(* Logix 5000 project; controller DispersionPlc vendor 1 type 14 code 108 rev 34.11; software revision 34.01; part 13 of 22 *)
(* tags used below, declared in another part *)
   Estop_Disp : ALIAS FOR Local:3:I.Data.1;
   Estop_Inx : ALIAS FOR Local:3:I.Data.3;
   FC_4305_xx : AStd_PIDInterface;
   FCV_4305 : ALIAS FOR Local:13:O.Ch0Data;
   FIT_4305_xx : AStd_AnalogInput;
   FIT_4305_xx_AOI : AStd_AI_AOI;
   FIT_4305_xx_Holding : DINT;
   FIT_4305_xx_Samples : DINT;
   FV_4305_xx : AStd_VlvModulating;
   FV_4305_xx_AOI : AStd_VlVModulating_AOI;
   K400_PhaseTransfer : AStd_PLI;
   K400_PhaseTransfer_AOI : AStd_PLI_AOI;
   K400_PhaseTransfer_StepComplete : BOOL[32];
   LS_28_H : TIMER;
   LS_28_H_Alarm : BOOL;
   LS_4302_High : BOOL;
   P_4305 : AStd_FVNR;
   P_4305_AOI : AStd_FVNR_AOI;
   PUMP_P_4305_AUX : ALIAS FOR Local:1:I.Data[1].7;
   PUMP_P_4305_RUN : ALIAS FOR Local:1:O.Data[0].7;
   RO_HE4305_PhaseROHotWaterDrop : AStd_PLI;
   RO_HE4305_PhaseROHotWaterDrop_AOI : AStd_PLI_AOI;
   RO_HE4305_PhaseROWaterAddition : AStd_PLI;
   RO_Preheat_Temp : DINT;
   T4301_T4302_Xfer_In_Enable_Ctrl : BOOL;
   TC_4305_1 : AStd_PIDInterface;
   TC_4305_1_AOI : AStd_PIDInterface_AOI;
   TC_4305_1_PID : PID_ENHANCED;
   TCV_4305_1 : AStd_VlvModulating;
   TCV_4305_1_AOI : AStd_VlVModulating_AOI;
   TIT_4305_1 : AStd_AnalogInput;
   TIT_4305_1_AOI : AStd_AI_AOI;
   TIT_K400_1 : AStd_AnalogInput;
   TIT_K400_3 : AStd_AnalogInput;
   WIT_4302_1 : AStd_AnalogInput;
   XV_4301_8 : AStd_VlvOC;
   XV_4301_8_AOI : AStd_VlvOC_AOI;
   XV_4301_8_IOpn : BOOL;
   XV_4301_8_OCls : BOOL;
   XV_4302_7 : AStd_VlvOC;
   XV_4302_8 : AStd_VlvOC;
   XV_4302_9 : AStd_VlvOC;
   XV_4306_3 : AStd_VlvOC;
   XV_4307_3 : AStd_VlvOC;
   XV_K400_6 : AStd_VlvOC;
   XV_K400_7 : AStd_VlvOC;
(* Unit_K400, continued *)

ROUTINE MainRoutine   (* ladder *)
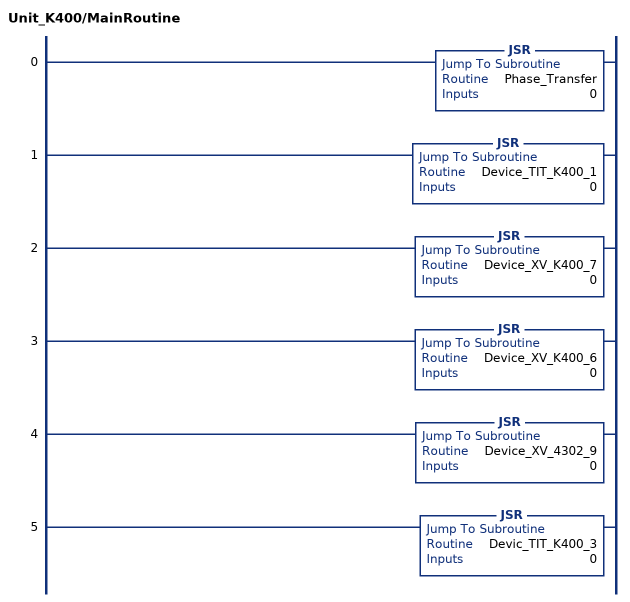
   0: JSR(Phase_Transfer,0);
   1: JSR(Device_TIT_K400_1,0);
   2: JSR(Device_XV_K400_7,0);
   3: JSR(Device_XV_K400_6,0);
   4: JSR(Device_XV_4302_9,0);
   5: JSR(Devic_TIT_K400_3,0);
END_ROUTINE

ROUTINE Phase_Transfer   (* ladder *)
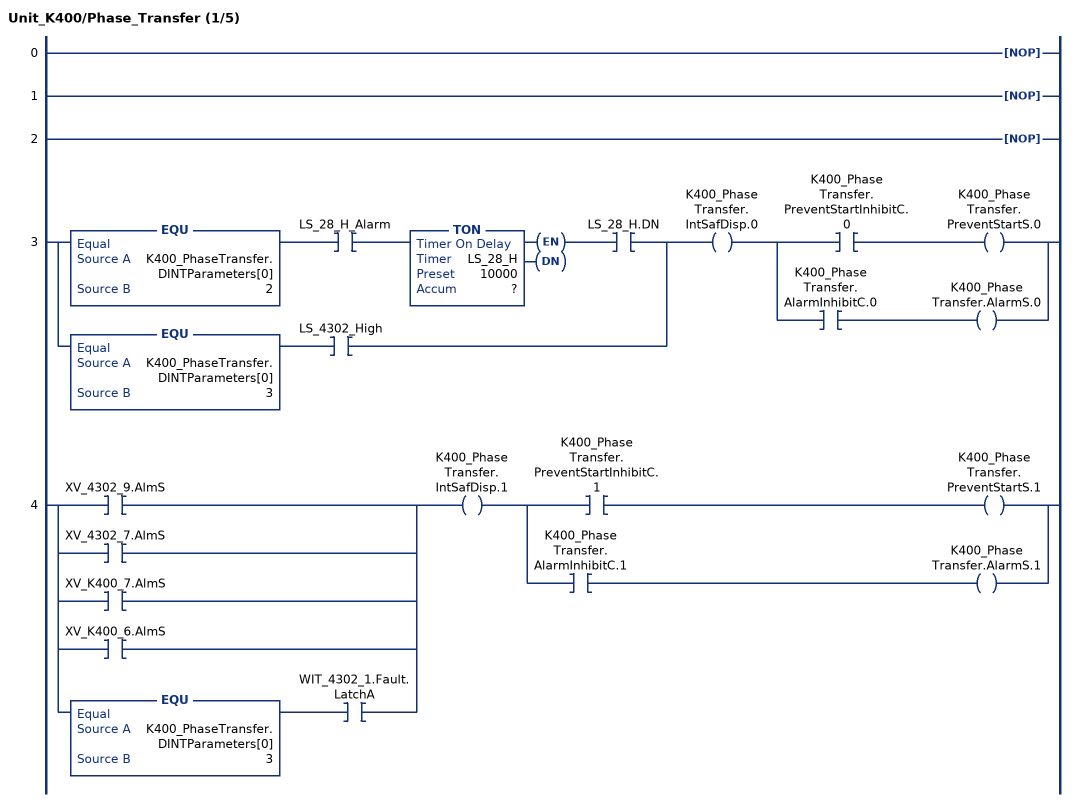
   0: NOP();
   1: NOP();
   2: NOP();
   3: [EQU(K400_PhaseTransfer.DINTParameters[0],2) XIC(LS_28_H_Alarm) TON(LS_28_H,?,?) XIC(LS_28_H.DN) ,EQU(K400_PhaseTransfer.DINTParameters[0],3) XIC(LS_4302_High) ]OTE(K400_PhaseTransfer.IntSafDisp.0)[XIC(K400_PhaseTransfer.PreventStartInhibitC.0) OTE(K400_PhaseTransfer.PreventStartS.0) ,XIC(K400_PhaseTransfer.AlarmInhibitC.0) OTE(K400_PhaseTransfer.AlarmS.0) ];
   4: [XIC(XV_4302_9.AlmS) ,XIC(XV_4302_7.AlmS) ,XIC(XV_K400_7.AlmS) ,XIC(XV_K400_6.AlmS) ,EQU(K400_PhaseTransfer.DINTParameters[0],3) XIC(WIT_4302_1.Fault.LatchA) ]OTE(K400_PhaseTransfer.IntSafDisp.1)[XIC(K400_PhaseTransfer.PreventStartInhibitC.1) OTE(K400_PhaseTransfer.PreventStartS.1) ,XIC(K400_PhaseTransfer.AlarmInhibitC.1) OTE(K400_PhaseTransfer.AlarmS.1) ];
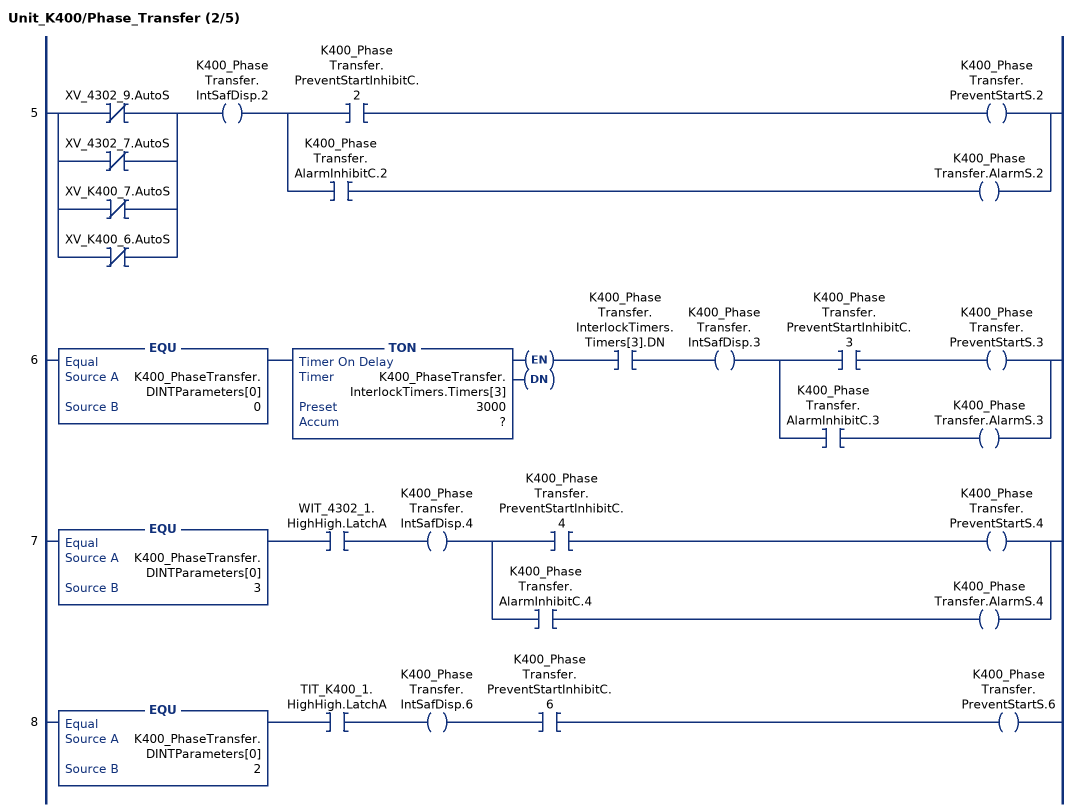
   5: [XIO(XV_4302_9.AutoS) ,XIO(XV_4302_7.AutoS) ,XIO(XV_K400_7.AutoS) ,XIO(XV_K400_6.AutoS) ]OTE(K400_PhaseTransfer.IntSafDisp.2)[XIC(K400_PhaseTransfer.PreventStartInhibitC.2) OTE(K400_PhaseTransfer.PreventStartS.2) ,XIC(K400_PhaseTransfer.AlarmInhibitC.2) OTE(K400_PhaseTransfer.AlarmS.2) ];
   6: EQU(K400_PhaseTransfer.DINTParameters[0],0)TON(K400_PhaseTransfer.InterlockTimers.Timers[3],?,?)XIC(K400_PhaseTransfer.InterlockTimers.Timers[3].DN)OTE(K400_PhaseTransfer.IntSafDisp.3)[XIC(K400_PhaseTransfer.PreventStartInhibitC.3) OTE(K400_PhaseTransfer.PreventStartS.3) ,XIC(K400_PhaseTransfer.AlarmInhibitC.3) OTE(K400_PhaseTransfer.AlarmS.3) ];
   7: EQU(K400_PhaseTransfer.DINTParameters[0],3)XIC(WIT_4302_1.HighHigh.LatchA)OTE(K400_PhaseTransfer.IntSafDisp.4)[XIC(K400_PhaseTransfer.PreventStartInhibitC.4) OTE(K400_PhaseTransfer.PreventStartS.4) ,XIC(K400_PhaseTransfer.AlarmInhibitC.4) OTE(K400_PhaseTransfer.AlarmS.4) ];
   8: EQU(K400_PhaseTransfer.DINTParameters[0],2)XIC(TIT_K400_1.HighHigh.LatchA)OTE(K400_PhaseTransfer.IntSafDisp.6)XIC(K400_PhaseTransfer.PreventStartInhibitC.6)OTE(K400_PhaseTransfer.PreventStartS.6);
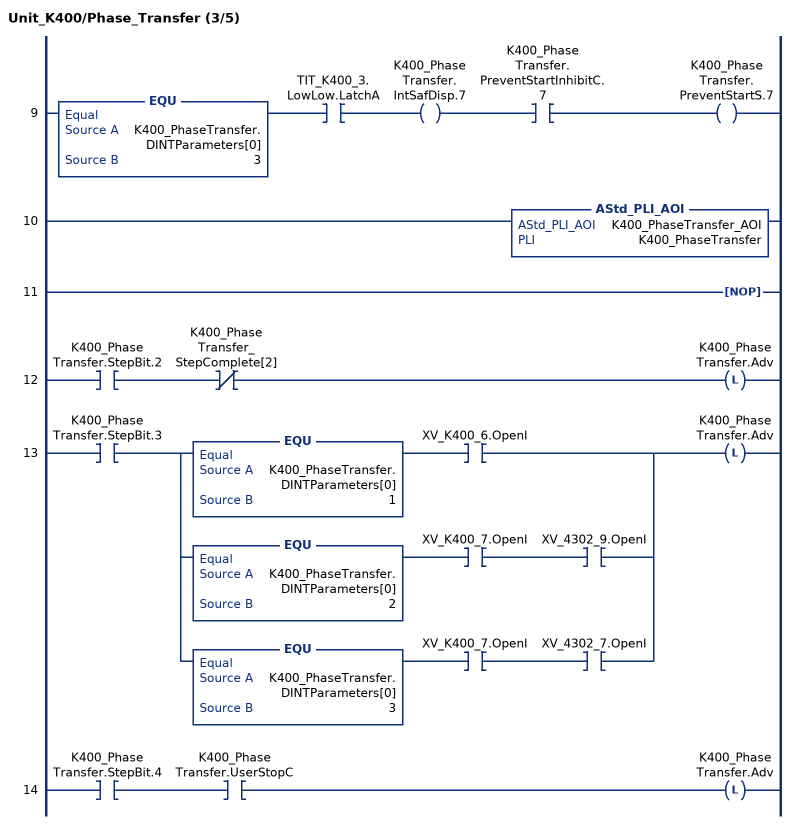
   9: EQU(K400_PhaseTransfer.DINTParameters[0],3)XIC(TIT_K400_3.LowLow.LatchA)OTE(K400_PhaseTransfer.IntSafDisp.7)XIC(K400_PhaseTransfer.PreventStartInhibitC.7)OTE(K400_PhaseTransfer.PreventStartS.7);
   10: AStd_PLI_AOI(K400_PhaseTransfer_AOI,K400_PhaseTransfer);
   11: NOP();
   12: XIC(K400_PhaseTransfer.StepBit.2)XIO(K400_PhaseTransfer_StepComplete[2])OTL(K400_PhaseTransfer.Adv);
   13: XIC(K400_PhaseTransfer.StepBit.3)[EQU(K400_PhaseTransfer.DINTParameters[0],1) XIC(XV_K400_6.OpenI) ,EQU(K400_PhaseTransfer.DINTParameters[0],2) XIC(XV_K400_7.OpenI) XIC(XV_4302_9.OpenI) ,EQU(K400_PhaseTransfer.DINTParameters[0],3) XIC(XV_K400_7.OpenI) XIC(XV_4302_7.OpenI) ]OTL(K400_PhaseTransfer.Adv);
   14: XIC(K400_PhaseTransfer.StepBit.4)XIC(K400_PhaseTransfer.UserStopC)OTL(K400_PhaseTransfer.Adv);
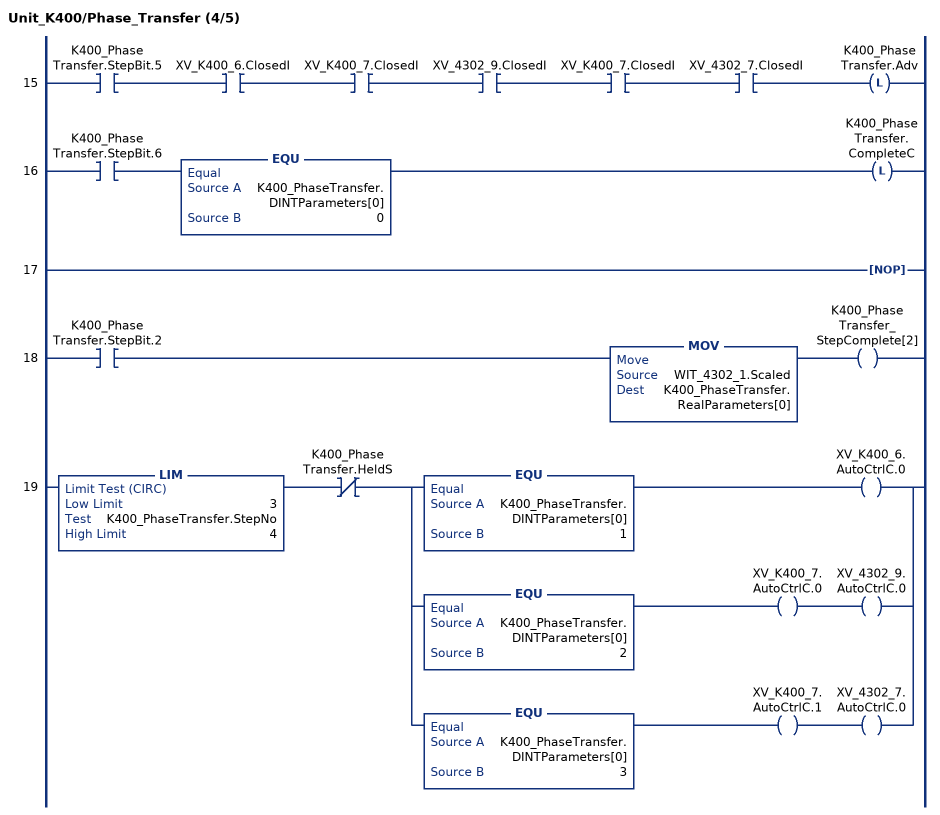
   15: XIC(K400_PhaseTransfer.StepBit.5)XIC(XV_K400_6.ClosedI)XIC(XV_K400_7.ClosedI)XIC(XV_4302_9.ClosedI)XIC(XV_K400_7.ClosedI)XIC(XV_4302_7.ClosedI)OTL(K400_PhaseTransfer.Adv);
   16: XIC(K400_PhaseTransfer.StepBit.6)EQU(K400_PhaseTransfer.DINTParameters[0],0)OTL(K400_PhaseTransfer.CompleteC);
   17: NOP();
   18: XIC(K400_PhaseTransfer.StepBit.2)MOV(WIT_4302_1.Scaled,K400_PhaseTransfer.RealParameters[0])OTE(K400_PhaseTransfer_StepComplete[2]);
   19: LIM(3,K400_PhaseTransfer.StepNo,4)XIO(K400_PhaseTransfer.HeldS)[EQU(K400_PhaseTransfer.DINTParameters[0],1) OTE(XV_K400_6.AutoCtrlC.0) ,EQU(K400_PhaseTransfer.DINTParameters[0],2) OTE(XV_K400_7.AutoCtrlC.0) OTE(XV_4302_9.AutoCtrlC.0) ,EQU(K400_PhaseTransfer.DINTParameters[0],3) OTE(XV_K400_7.AutoCtrlC.1) OTE(XV_4302_7.AutoCtrlC.0) ];
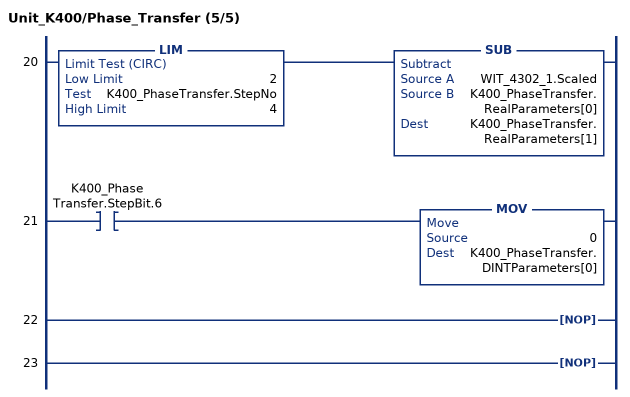
   20: LIM(2,K400_PhaseTransfer.StepNo,4)SUB(WIT_4302_1.Scaled,K400_PhaseTransfer.RealParameters[0],K400_PhaseTransfer.RealParameters[1]);
   21: XIC(K400_PhaseTransfer.StepBit.6)MOV(0,K400_PhaseTransfer.DINTParameters[0]);
   22: NOP();
   23: NOP();
END_ROUTINE
END_PROGRAM

PROGRAM Unit_RO_HE4305   (* main routine MainRoutine *)
VAR
   Totalizers : REAL[10];
END_VAR

ROUTINE Device_FIT_4305_xx   (* ladder *)
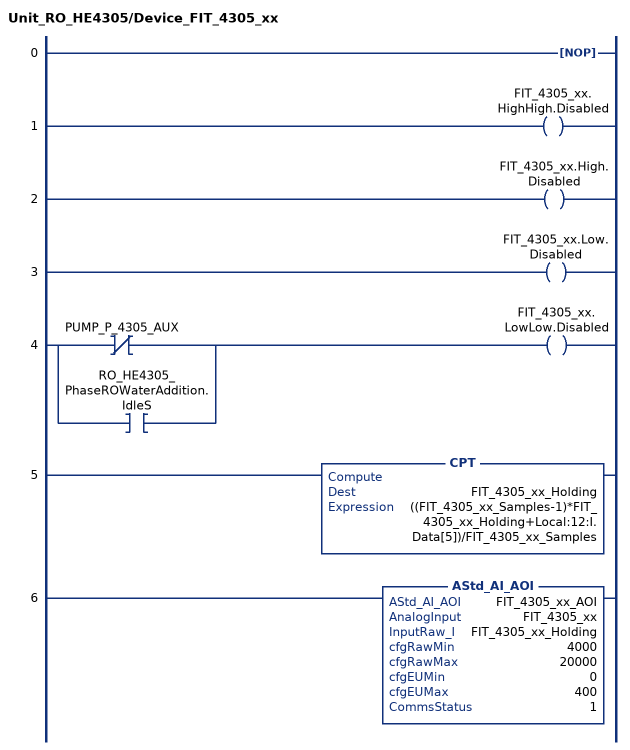
   0: NOP();
   1: OTE(FIT_4305_xx.HighHigh.Disabled);
   2: OTE(FIT_4305_xx.High.Disabled);
   3: OTE(FIT_4305_xx.Low.Disabled);
   4: [XIO(PUMP_P_4305_AUX) ,XIC(RO_HE4305_PhaseROWaterAddition.IdleS) ]OTE(FIT_4305_xx.LowLow.Disabled);
   5: CPT(FIT_4305_xx_Holding,((FIT_4305_xx_Samples-1)*FIT_4305_xx_Holding+Local:12:I.Data[5])/FIT_4305_xx_Samples);
   6: AStd_AI_AOI(FIT_4305_xx_AOI,FIT_4305_xx,FIT_4305_xx_Holding,4000,20000,0,400,1);
END_ROUTINE

ROUTINE Device_FV_4305_xx   (* ladder *)
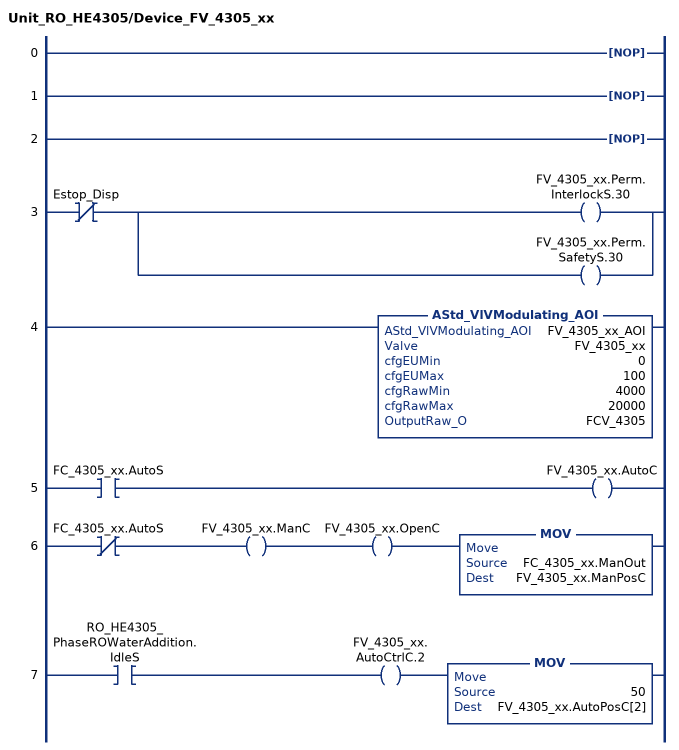
   0: NOP();
   1: NOP();
   2: NOP();
   3: XIO(Estop_Disp)[OTE(FV_4305_xx.Perm.InterlockS.30) ,OTE(FV_4305_xx.Perm.SafetyS.30) ];
   4: AStd_VlVModulating_AOI(FV_4305_xx_AOI,FV_4305_xx,0,100,4000,20000,FCV_4305);
   5: XIC(FC_4305_xx.AutoS)OTE(FV_4305_xx.AutoC);
   6: XIO(FC_4305_xx.AutoS)OTE(FV_4305_xx.ManC)OTE(FV_4305_xx.OpenC)MOV(FC_4305_xx.ManOut,FV_4305_xx.ManPosC);
   7: XIC(RO_HE4305_PhaseROWaterAddition.IdleS)OTE(FV_4305_xx.AutoCtrlC.2)MOV(50,FV_4305_xx.AutoPosC[2]);
END_ROUTINE

ROUTINE Device_P_4305   (* ladder *)
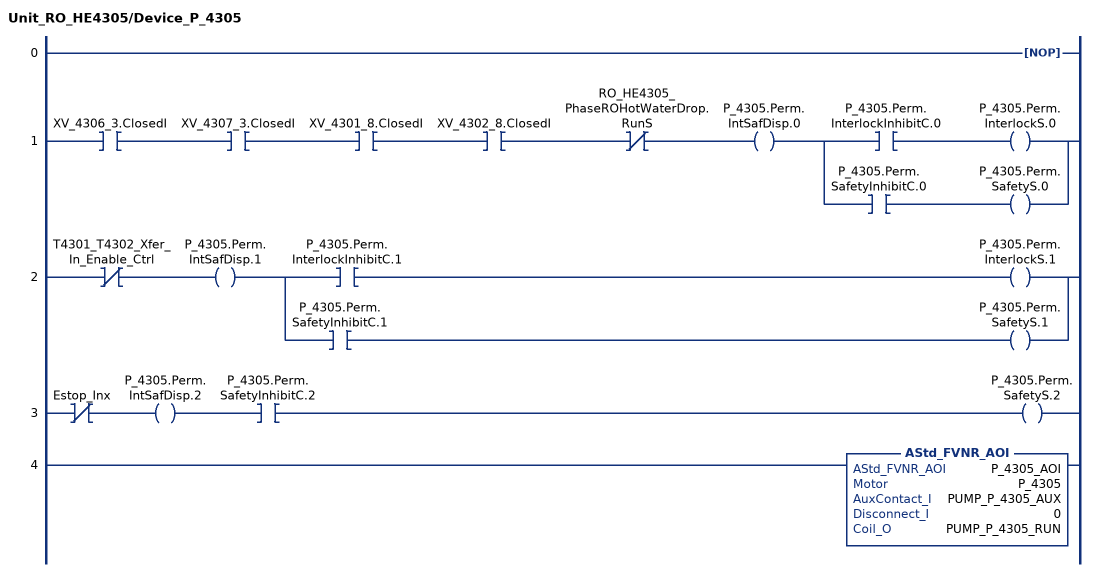
   0: NOP();
   1: XIC(XV_4306_3.ClosedI)XIC(XV_4307_3.ClosedI)XIC(XV_4301_8.ClosedI)XIC(XV_4302_8.ClosedI)XIO(RO_HE4305_PhaseROHotWaterDrop.RunS)OTE(P_4305.Perm.IntSafDisp.0)[XIC(P_4305.Perm.InterlockInhibitC.0) OTE(P_4305.Perm.InterlockS.0) ,XIC(P_4305.Perm.SafetyInhibitC.0) OTE(P_4305.Perm.SafetyS.0) ];
   2: XIO(T4301_T4302_Xfer_In_Enable_Ctrl)OTE(P_4305.Perm.IntSafDisp.1)[XIC(P_4305.Perm.InterlockInhibitC.1) OTE(P_4305.Perm.InterlockS.1) ,XIC(P_4305.Perm.SafetyInhibitC.1) OTE(P_4305.Perm.SafetyS.1) ];
   3: XIO(Estop_Inx)OTE(P_4305.Perm.IntSafDisp.2)XIC(P_4305.Perm.SafetyInhibitC.2)OTE(P_4305.Perm.SafetyS.2);
   4: AStd_FVNR_AOI(P_4305_AOI,P_4305,PUMP_P_4305_AUX,0,PUMP_P_4305_RUN);
END_ROUTINE

ROUTINE Device_TCV_4305_1   (* ladder *)
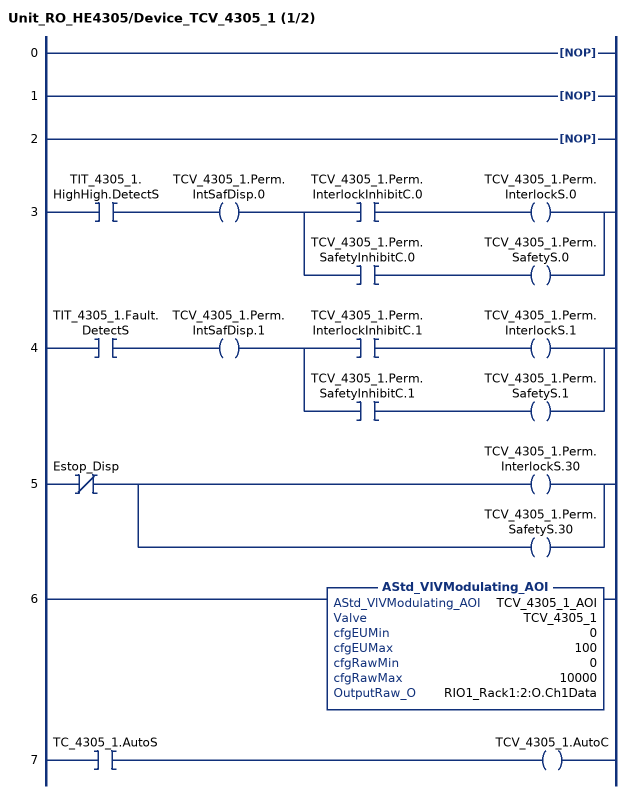
   0: NOP();
   1: NOP();
   2: NOP();
   3: XIC(TIT_4305_1.HighHigh.DetectS)OTE(TCV_4305_1.Perm.IntSafDisp.0)[XIC(TCV_4305_1.Perm.InterlockInhibitC.0) OTE(TCV_4305_1.Perm.InterlockS.0) ,XIC(TCV_4305_1.Perm.SafetyInhibitC.0) OTE(TCV_4305_1.Perm.SafetyS.0) ];
   4: XIC(TIT_4305_1.Fault.DetectS)OTE(TCV_4305_1.Perm.IntSafDisp.1)[XIC(TCV_4305_1.Perm.InterlockInhibitC.1) OTE(TCV_4305_1.Perm.InterlockS.1) ,XIC(TCV_4305_1.Perm.SafetyInhibitC.1) OTE(TCV_4305_1.Perm.SafetyS.1) ];
   5: XIO(Estop_Disp)[OTE(TCV_4305_1.Perm.InterlockS.30) ,OTE(TCV_4305_1.Perm.SafetyS.30) ];
   6: AStd_VlVModulating_AOI(TCV_4305_1_AOI,TCV_4305_1,0,100,0,10000,RIO1_Rack1:2:O.Ch1Data);
   7: XIC(TC_4305_1.AutoS)OTE(TCV_4305_1.AutoC);
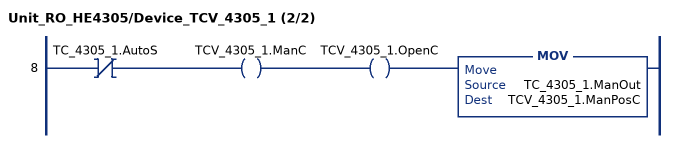
   8: XIO(TC_4305_1.AutoS)OTE(TCV_4305_1.ManC)OTE(TCV_4305_1.OpenC)MOV(TC_4305_1.ManOut,TCV_4305_1.ManPosC);
END_ROUTINE

ROUTINE Device_TIT_4305_1   (* ladder *)
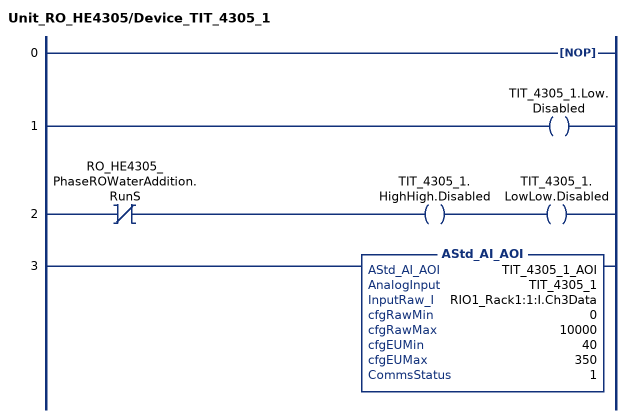
   0: NOP();
   1: OTE(TIT_4305_1.Low.Disabled);
   2: XIO(RO_HE4305_PhaseROWaterAddition.RunS)OTE(TIT_4305_1.HighHigh.Disabled)OTE(TIT_4305_1.LowLow.Disabled);
   3: AStd_AI_AOI(TIT_4305_1_AOI,TIT_4305_1,RIO1_Rack1:1:I.Ch3Data,0,10000,40,350,1);
END_ROUTINE

ROUTINE Device_XV_4301_8   (* ladder *)
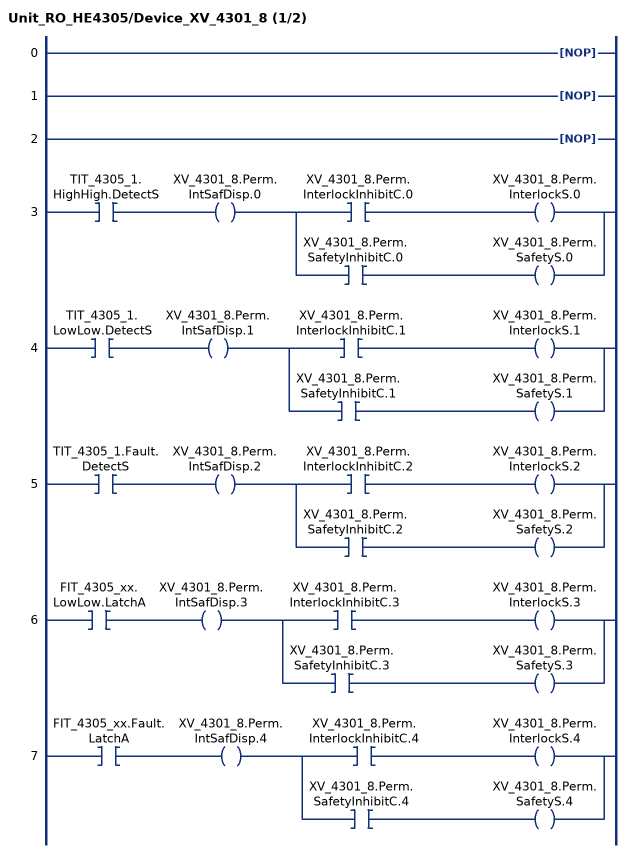
   0: NOP();
   1: NOP();
   2: NOP();
   3: XIC(TIT_4305_1.HighHigh.DetectS)OTE(XV_4301_8.Perm.IntSafDisp.0)[XIC(XV_4301_8.Perm.InterlockInhibitC.0) OTE(XV_4301_8.Perm.InterlockS.0) ,XIC(XV_4301_8.Perm.SafetyInhibitC.0) OTE(XV_4301_8.Perm.SafetyS.0) ];
   4: XIC(TIT_4305_1.LowLow.DetectS)OTE(XV_4301_8.Perm.IntSafDisp.1)[XIC(XV_4301_8.Perm.InterlockInhibitC.1) OTE(XV_4301_8.Perm.InterlockS.1) ,XIC(XV_4301_8.Perm.SafetyInhibitC.1) OTE(XV_4301_8.Perm.SafetyS.1) ];
   5: XIC(TIT_4305_1.Fault.DetectS)OTE(XV_4301_8.Perm.IntSafDisp.2)[XIC(XV_4301_8.Perm.InterlockInhibitC.2) OTE(XV_4301_8.Perm.InterlockS.2) ,XIC(XV_4301_8.Perm.SafetyInhibitC.2) OTE(XV_4301_8.Perm.SafetyS.2) ];
   6: XIC(FIT_4305_xx.LowLow.LatchA)OTE(XV_4301_8.Perm.IntSafDisp.3)[XIC(XV_4301_8.Perm.InterlockInhibitC.3) OTE(XV_4301_8.Perm.InterlockS.3) ,XIC(XV_4301_8.Perm.SafetyInhibitC.3) OTE(XV_4301_8.Perm.SafetyS.3) ];
   7: XIC(FIT_4305_xx.Fault.LatchA)OTE(XV_4301_8.Perm.IntSafDisp.4)[XIC(XV_4301_8.Perm.InterlockInhibitC.4) OTE(XV_4301_8.Perm.InterlockS.4) ,XIC(XV_4301_8.Perm.SafetyInhibitC.4) OTE(XV_4301_8.Perm.SafetyS.4) ];
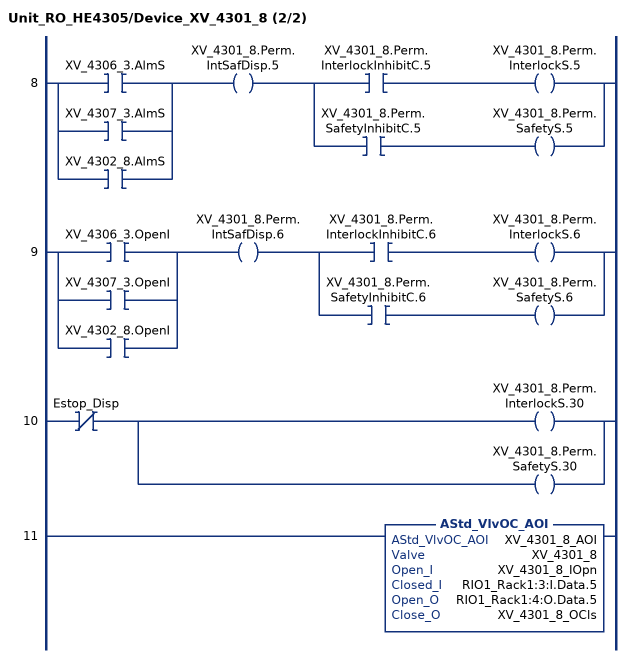
   8: [XIC(XV_4306_3.AlmS) ,XIC(XV_4307_3.AlmS) ,XIC(XV_4302_8.AlmS) ]OTE(XV_4301_8.Perm.IntSafDisp.5)[XIC(XV_4301_8.Perm.InterlockInhibitC.5) OTE(XV_4301_8.Perm.InterlockS.5) ,XIC(XV_4301_8.Perm.SafetyInhibitC.5) OTE(XV_4301_8.Perm.SafetyS.5) ];
   9: [XIC(XV_4306_3.OpenI) ,XIC(XV_4307_3.OpenI) ,XIC(XV_4302_8.OpenI) ]OTE(XV_4301_8.Perm.IntSafDisp.6)[XIC(XV_4301_8.Perm.InterlockInhibitC.6) OTE(XV_4301_8.Perm.InterlockS.6) ,XIC(XV_4301_8.Perm.SafetyInhibitC.6) OTE(XV_4301_8.Perm.SafetyS.6) ];
   10: XIO(Estop_Disp)[OTE(XV_4301_8.Perm.InterlockS.30) ,OTE(XV_4301_8.Perm.SafetyS.30) ];
   11: AStd_VlvOC_AOI(XV_4301_8_AOI,XV_4301_8,XV_4301_8_IOpn,RIO1_Rack1:3:I.Data.5,RIO1_Rack1:4:O.Data.5,XV_4301_8_OCls);
END_ROUTINE

ROUTINE MainRoutine   (* ladder *)
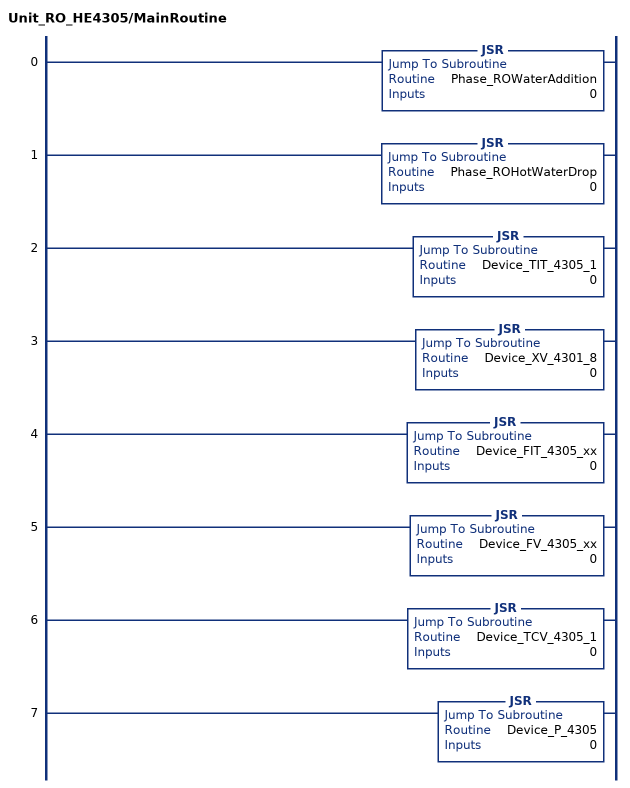
   0: JSR(Phase_ROWaterAddition,0);
   1: JSR(Phase_ROHotWaterDrop,0);
   2: JSR(Device_TIT_4305_1,0);
   3: JSR(Device_XV_4301_8,0);
   4: JSR(Device_FIT_4305_xx,0);
   5: JSR(Device_FV_4305_xx,0);
   6: JSR(Device_TCV_4305_1,0);
   7: JSR(Device_P_4305,0);
END_ROUTINE

ROUTINE Phase_ROHotWaterDrop   (* ladder *)
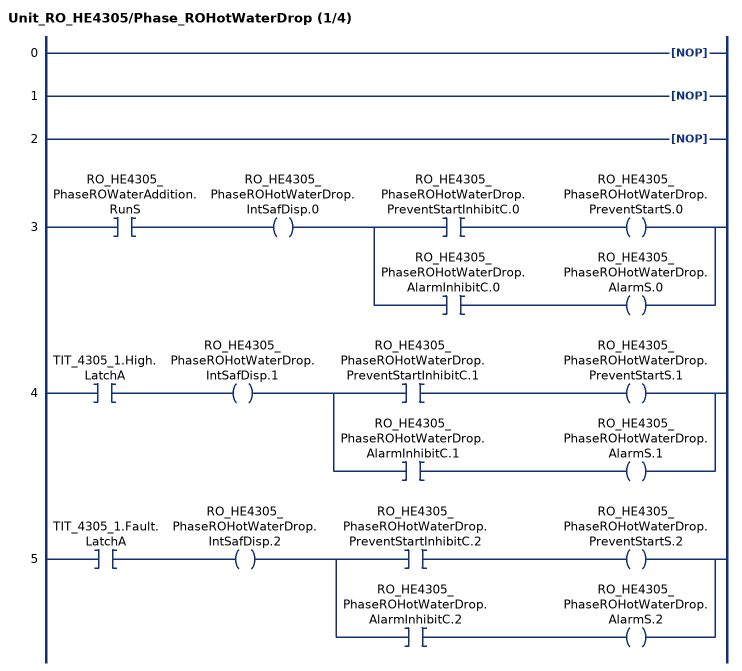
   0: NOP();
   1: NOP();
   2: NOP();
   3: XIC(RO_HE4305_PhaseROWaterAddition.RunS)OTE(RO_HE4305_PhaseROHotWaterDrop.IntSafDisp.0)[XIC(RO_HE4305_PhaseROHotWaterDrop.PreventStartInhibitC.0) OTE(RO_HE4305_PhaseROHotWaterDrop.PreventStartS.0) ,XIC(RO_HE4305_PhaseROHotWaterDrop.AlarmInhibitC.0) OTE(RO_HE4305_PhaseROHotWaterDrop.AlarmS.0) ];
   4: XIC(TIT_4305_1.High.LatchA)OTE(RO_HE4305_PhaseROHotWaterDrop.IntSafDisp.1)[XIC(RO_HE4305_PhaseROHotWaterDrop.PreventStartInhibitC.1) OTE(RO_HE4305_PhaseROHotWaterDrop.PreventStartS.1) ,XIC(RO_HE4305_PhaseROHotWaterDrop.AlarmInhibitC.1) OTE(RO_HE4305_PhaseROHotWaterDrop.AlarmS.1) ];
   5: XIC(TIT_4305_1.Fault.LatchA)OTE(RO_HE4305_PhaseROHotWaterDrop.IntSafDisp.2)[XIC(RO_HE4305_PhaseROHotWaterDrop.PreventStartInhibitC.2) OTE(RO_HE4305_PhaseROHotWaterDrop.PreventStartS.2) ,XIC(RO_HE4305_PhaseROHotWaterDrop.AlarmInhibitC.2) OTE(RO_HE4305_PhaseROHotWaterDrop.AlarmS.2) ];
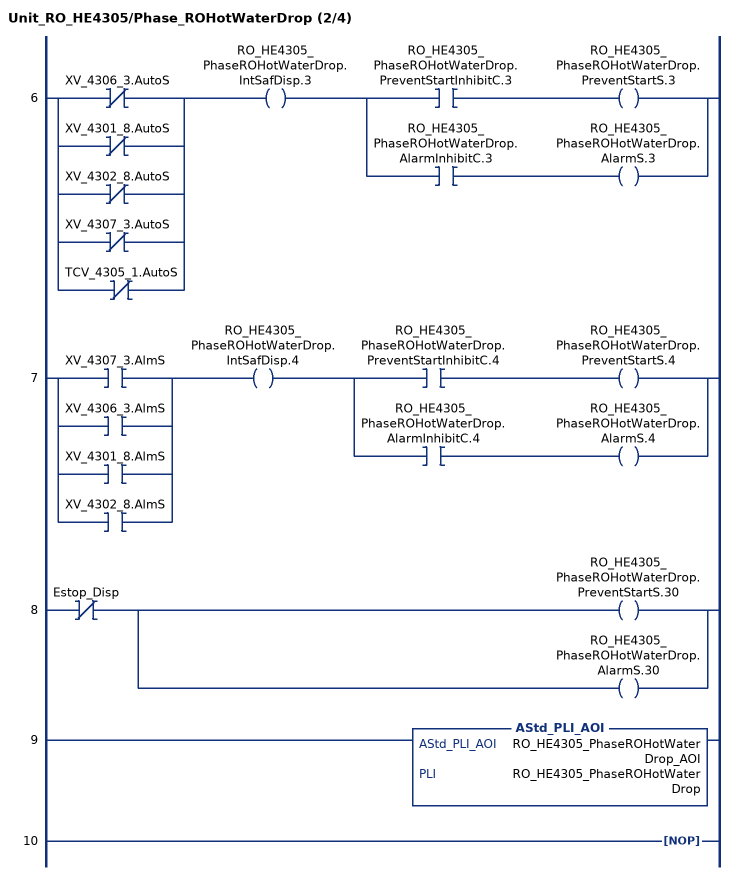
   6: [XIO(XV_4306_3.AutoS) ,XIO(XV_4301_8.AutoS) ,XIO(XV_4302_8.AutoS) ,XIO(XV_4307_3.AutoS) ,XIO(TCV_4305_1.AutoS) ]OTE(RO_HE4305_PhaseROHotWaterDrop.IntSafDisp.3)[XIC(RO_HE4305_PhaseROHotWaterDrop.PreventStartInhibitC.3) OTE(RO_HE4305_PhaseROHotWaterDrop.PreventStartS.3) ,XIC(RO_HE4305_PhaseROHotWaterDrop.AlarmInhibitC.3) OTE(RO_HE4305_PhaseROHotWaterDrop.AlarmS.3) ];
   7: [XIC(XV_4307_3.AlmS) ,XIC(XV_4306_3.AlmS) ,XIC(XV_4301_8.AlmS) ,XIC(XV_4302_8.AlmS) ]OTE(RO_HE4305_PhaseROHotWaterDrop.IntSafDisp.4)[XIC(RO_HE4305_PhaseROHotWaterDrop.PreventStartInhibitC.4) OTE(RO_HE4305_PhaseROHotWaterDrop.PreventStartS.4) ,XIC(RO_HE4305_PhaseROHotWaterDrop.AlarmInhibitC.4) OTE(RO_HE4305_PhaseROHotWaterDrop.AlarmS.4) ];
   8: XIO(Estop_Disp)[OTE(RO_HE4305_PhaseROHotWaterDrop.PreventStartS.30) ,OTE(RO_HE4305_PhaseROHotWaterDrop.AlarmS.30) ];
   9: AStd_PLI_AOI(RO_HE4305_PhaseROHotWaterDrop_AOI,RO_HE4305_PhaseROHotWaterDrop);
   10: NOP();
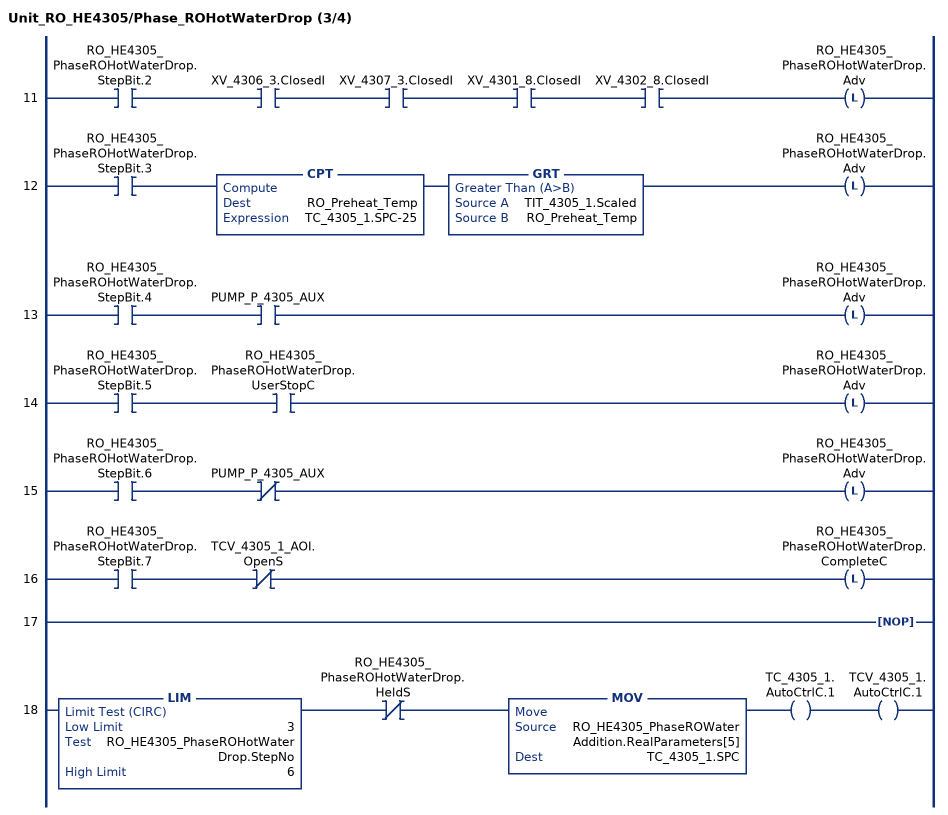
   11: XIC(RO_HE4305_PhaseROHotWaterDrop.StepBit.2)XIC(XV_4306_3.ClosedI)XIC(XV_4307_3.ClosedI)XIC(XV_4301_8.ClosedI)XIC(XV_4302_8.ClosedI)OTL(RO_HE4305_PhaseROHotWaterDrop.Adv);
   12: XIC(RO_HE4305_PhaseROHotWaterDrop.StepBit.3)CPT(RO_Preheat_Temp,TC_4305_1.SPC-25)GRT(TIT_4305_1.Scaled,RO_Preheat_Temp)OTL(RO_HE4305_PhaseROHotWaterDrop.Adv);
   13: XIC(RO_HE4305_PhaseROHotWaterDrop.StepBit.4)XIC(PUMP_P_4305_AUX)OTL(RO_HE4305_PhaseROHotWaterDrop.Adv);
   14: XIC(RO_HE4305_PhaseROHotWaterDrop.StepBit.5)XIC(RO_HE4305_PhaseROHotWaterDrop.UserStopC)OTL(RO_HE4305_PhaseROHotWaterDrop.Adv);
   15: XIC(RO_HE4305_PhaseROHotWaterDrop.StepBit.6)XIO(PUMP_P_4305_AUX)OTL(RO_HE4305_PhaseROHotWaterDrop.Adv);
   16: XIC(RO_HE4305_PhaseROHotWaterDrop.StepBit.7)XIO(TCV_4305_1_AOI.OpenS)OTL(RO_HE4305_PhaseROHotWaterDrop.CompleteC);
   17: NOP();
   18: LIM(3,RO_HE4305_PhaseROHotWaterDrop.StepNo,6)XIO(RO_HE4305_PhaseROHotWaterDrop.HeldS)MOV(RO_HE4305_PhaseROWaterAddition.RealParameters[5],TC_4305_1.SPC)OTE(TC_4305_1.AutoCtrlC.1)OTE(TCV_4305_1.AutoCtrlC.1);
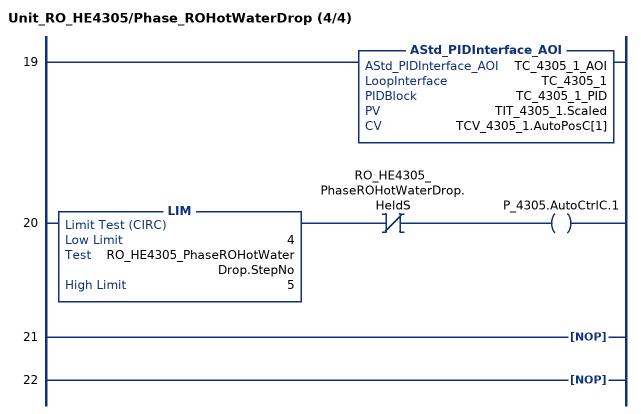
   19: AStd_PIDInterface_AOI(TC_4305_1_AOI,TC_4305_1,TC_4305_1_PID,TIT_4305_1.Scaled,TCV_4305_1.AutoPosC[1]);
   20: LIM(4,RO_HE4305_PhaseROHotWaterDrop.StepNo,5)XIO(RO_HE4305_PhaseROHotWaterDrop.HeldS)OTE(P_4305.AutoCtrlC.1);
   21: NOP();
   22: NOP();
END_ROUTINE
